FUNCTION_BLOCK AccumTimes
VAR_INPUT
	State: BOOL;	
END_VAR

VAR PERSISTENT
	Num : WORD;
	ResetAccum: BOOL;

	cntOn: CTU;
	Accum: AccumDDHHMM;
	On: AccumDDHHMM;
	Off: AccumDDHHMM;
END_VAR

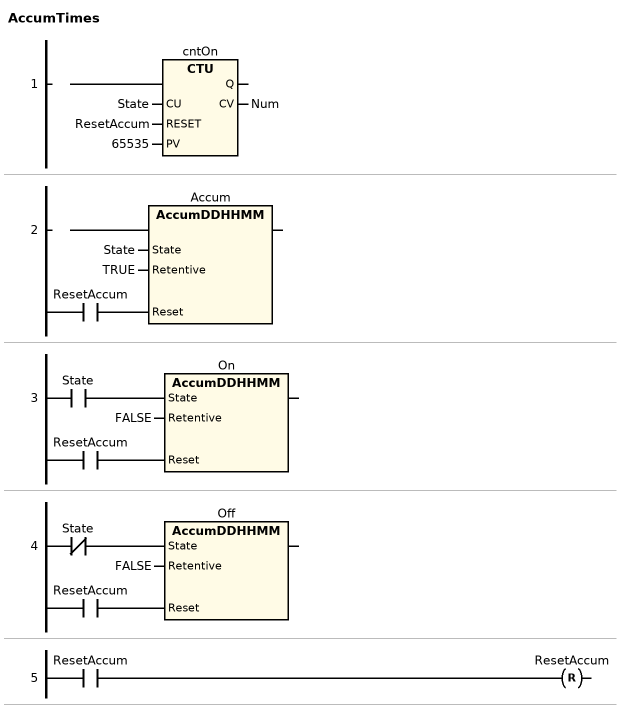
// NETWORK 1
cntOn(CU := State, RESET := ResetAccum, PV := 65535, CV => Num); // CTU

// NETWORK 2
Accum(State := State, Retentive := TRUE, Reset := ResetAccum); // AccumDDHHMM

// NETWORK 3
On(State := State, Retentive := FALSE, Reset := ResetAccum); // AccumDDHHMM

// NETWORK 4
Off(State := NOT State, Retentive := FALSE, Reset := ResetAccum); // AccumDDHHMM

// NETWORK 5
ResetAccum R= ResetAccum;

END_FUNCTION_BLOCK

(* stored: Version 1.1.0.1, ProductVersion 3.1.4024.12
   POU AccumTimes: Id {374117b7-f183-496f-8247-5eaf7ba27164}, SpecialFunc None *)
